TYPE ST_FlowConfig :
STRUCT
	sName : STRING(255);
	aChannelConfigs : ARRAY[0..SiftClientParameters.MAX_NUM_CHANNELS_PER_FLOW - 1] OF ST_ChannelConfig;
	nNumChannelConfigs : UDINT;
END_STRUCT
END_TYPE

(* stored: Version 1.1.0.1
   DUT ST_FlowConfig: Id {d7b905d6-4a1e-4014-9e1a-01f024836dbe} *)
